FUNCTION_BLOCK Test_TStreamAdd_Read_PVOID EXTENDS T_UnitTestBase
VAR
    Stream : T_Stream(StreamLength := 2);
    Bob : INT;
END_VAR



Stream.Init(2);

Stream.Add_PVOID(ADR(Bob));
    
Assertion.AssertEquals_UDINT(
    Expected :=8,
    Actual := Stream.Position,
    VariableName := 'Stream.Position');
    
Stream.Seek(0);

Assertion.AssertEquals_PVOID(
    Expected := ADR(Bob),
    Actual := Stream.Read_PVOID(),
    VariableName := 'Stream.Read_PVOID()');
    
Assertion.AssertEquals_UDINT(
    Expected := 8,
    Actual := Stream.Position,
    VariableName := 'Stream.Position');
    
    
TestFinished();

END_FUNCTION_BLOCK

(* stored: Version 1.1.0.1, ProductVersion 3.1.4024.4
   POU Test_TStreamAdd_Read_PVOID: Id {84951354-6441-44c9-b63c-255267689420}, SpecialFunc None *)
